{attribute 'call_after_init'}
FUNCTION_BLOCK FINAL DintParam EXTENDS BaseParam
VAR_INPUT
END_VAR
VAR_OUTPUT
	value: DINT;
END_VAR
VAR
	
END_VAR

METHOD Change_Param
VAR_INPUT
	value	: STRING;
END_VAR
THIS^.value := STRING_TO_DINT(value);
_display := DINT_TO_STRING(THIS^.value);
END_METHOD

METHOD Quick_Change
VAR_INPUT
	value: DINT;
END_VAR
THIS^.value := value;
_display := DINT_TO_STRING(THIS^.value);
END_METHOD

END_FUNCTION_BLOCK

(* stored: Version 1.1.0.1, ProductVersion 3.1.4024.12
   POU DintParam: Id {764c489c-9bcf-42bf-b434-4a4c54212710}, SpecialFunc None
   Method Change_Param: Id {970f1f81-83a6-4d58-b98c-4eba7d8f35d2}
   Method Quick_Change: Id {86a06d80-8bab-44a4-9dcd-36eb09509be9} *)
